Yaskawa INFORM job: R1_W03,5,7(0,0)OK-KM.JBI

/JOB
//NAME R1_W03,5,7(0,0)OK-KM
///FOLDERNAME SCIANA-NOWY-R2-KM
//POS
///NPOS 93,93,0,4,0,0
///TOOL 0
///POSTYPE PULSE
///PULSE
C00000=97801,-92951,-68020,42573,91743,-12282
C00001=188064,-59139,-49719,51220,48350,-5801
C00002=182482,-29523,-13831,58220,47542,-10694
C00003=186503,-14327,-833,57181,45005,-9773
C00004=186887,-13436,-157,57022,44797,-9650
C00005=187358,-18276,-5525,56185,44980,-9089
C00006=193250,-27913,-6363,58294,38967,-9969
C00007=199995,-16364,1412,54222,35645,-7165
C00008=199327,-15584,1994,54497,36056,-7364
C00009=199882,-17213,782,54333,35681,-7234
C00010=195511,-15034,9725,61255,35872,-11434
C00011=195511,-14418,11078,61887,35615,-11785
C00012=194782,-15937,9357,61766,36202,-11793
C00013=185148,-27392,-13403,56780,46393,-9588
C00014=194611,-49573,-33459,572,31924,-22077
C00015=195793,-42632,-27790,-753,32004,-21336
C00016=196651,-38308,-23003,-1749,31294,-20781
C00017=197052,-37261,-22343,-2197,31434,-20529
C00018=196235,-39864,-25459,-1248,31997,-21059
C00019=202582,-39238,-15691,-30047,22851,-6468
C00020=202582,-38747,-14553,-30589,22461,-6206
C00021=199520,-48265,-22642,-26019,21519,-8620
C00022=195597,-45769,-34616,8656,41829,-26358
C00023=205752,-37498,-18561,-12983,36783,-12907
C00024=204602,-36516,-17940,-11961,36728,-13544
C00025=195976,-39153,-18531,9623,35365,-26897
C00026=197793,-59286,-35313,7977,35152,-25873
C00027=213331,-48054,-41686,15165,61809,3623
C00028=205738,-19523,-29471,74829,71236,32232
C00029=212963,6142,-9202,90968,67126,41175
C00030=215317,9223,-6508,90706,65425,41155
C00031=216300,10496,-4975,90717,64708,41017
C00032=216595,12699,-3002,90716,64489,40979
C00033=216298,10454,-5417,90600,64716,41144
C00034=215808,9900,10687,95987,67227,42354
C00035=216745,9111,9989,96016,66542,42343
C00036=217921,4618,-10524,75178,67269,44249
C00037=217494,5264,-8626,75589,67333,43807
C00038=217735,7158,-6190,75755,67018,43579
C00039=220892,-10252,-22721,78838,53086,40871
C00040=217823,-16385,-27408,79730,55193,40452
C00041=213331,-48054,-41686,15165,61809,3623
C00042=211970,-37779,-14430,6801,34223,17849
C00043=210033,-36470,-13605,8545,34568,16753
C00044=209079,-35786,-13170,9389,34755,16221
C00045=208450,-36922,-14985,9824,35355,15936
C00046=209854,-36909,-13406,8784,34242,16610
C00047=205470,-32937,-11332,12488,35564,14251
C00048=204626,-32211,-10856,14325,36093,12193
C00049=199934,-27052,-7307,22881,40247,-2541
C00050=194869,-21825,-3734,26674,42807,-10107
C00051=213331,-48054,-41686,15165,61809,3623
C00052=227546,10998,5486,35197,58444,-54182
C00053=229778,13536,7768,34321,57451,-53482
C00054=230708,14716,8755,33927,57078,-53172
C00055=230020,15168,9251,34245,57291,-53423
C00056=230799,13170,6502,33684,57536,-52967
C00057=230268,3975,-668,31886,61076,-53028
C00058=230588,3390,-1036,31786,60892,-52943
C00059=229243,2878,-1594,32267,61468,-53362
C00060=231252,-39648,-4608,102791,21542,-67561
C00061=237258,-22465,5967,96694,21446,-64692
C00062=234738,-18513,13230,101595,23495,-67322
C00063=234315,-17869,14270,102096,23835,-67616
C00064=232289,-15111,19504,104909,25555,-69249
C00065=228307,-22326,11440,100405,28029,-67502
C00066=226911,810,-3337,33104,62378,-54110
C00067=213331,-48054,-41686,15165,61809,3623
C00068=211661,-57251,-25562,-55725,28615,-3338
C00069=209733,-56166,-24995,-54213,27635,-4283
C00070=209042,-55506,-24648,-53560,27321,-4674
C00071=207937,-56864,-25063,-53502,26430,-4804
C00072=210138,-56838,-26044,-54013,28046,-4347
C00073=213122,-57928,-25912,-64752,31046,-795
C00074=213758,-58111,-26008,-65027,31436,-589
C00075=219568,-60488,-27163,-67374,34939,1257
C00076=220810,-61245,-27594,-67808,35688,1626
C00077=221756,-61566,-27753,-68083,36274,1881
C00078=225369,-69260,-37480,-66382,39447,1288
C00079=205312,-39468,-16273,-14091,10779,-39550
C00080=202035,-29821,-9269,-1691,11105,-45367
C00081=201708,-29499,-9054,-507,11133,-45924
C00082=202005,-28855,-8724,-1550,11270,-45435
C00083=201579,-30109,-10785,-40,11885,-46143
C00084=201147,-30171,-8613,1607,10520,-46916
C00085=197038,-23502,-5168,15044,12246,-53254
C00086=191968,-16947,-326,28829,13963,-59823
C00087=192443,-23943,-5231,28759,13289,-59765
C00088=194260,-31922,-10655,25195,12023,-58034
C00089=194296,-50223,-21768,31420,9737,-60851
C00090=140544,-88669,-51716,31420,85002,-60851
C00091=29274,49299,-4686,19206,94492,-76966
C00092=-18103,108044,15339,14006,98532,-83827
BC00000=366006,1190719,810332
BC00001=395488,1192063,911452
BC00002=367626,1192063,911456
BC00003=367626,1192063,911456
BC00004=367626,1192063,911456
BC00005=367626,1192063,911456
BC00006=367626,1192063,911456
BC00007=367626,1192063,911456
BC00008=367626,1192063,911456
BC00009=367626,1192063,911456
BC00010=367626,1192063,911456
BC00011=367626,1192063,911456
BC00012=367626,1192063,911456
BC00013=367626,1192063,911456
BC00014=339752,1192063,946029
BC00015=339752,1192063,946029
BC00016=339752,1192063,946029
BC00017=339752,1192063,946029
BC00018=339752,1192063,946029
BC00019=339752,1192063,946029
BC00020=339752,1192063,946029
BC00021=339752,1192063,946029
BC00022=339752,1192063,946029
BC00023=339752,1192063,946029
BC00024=339752,1192063,946029
BC00025=339752,1192063,946029
BC00026=339752,1192063,946029
BC00027=343711,1192063,995389
BC00028=386489,1191732,674467
BC00029=396646,1191635,580346
BC00030=396646,1192063,571372
BC00031=396646,1192063,567782
BC00032=396646,1192063,567782
BC00033=396646,1192063,567782
BC00034=396646,1192063,632887
BC00035=396646,1192063,632887
BC00036=396646,1192063,632887
BC00037=396646,1192063,632887
BC00038=396646,1192063,632887
BC00039=396646,1192063,584688
BC00040=396646,1192063,601373
BC00041=343711,1192063,995389
BC00042=340575,1192063,995049
BC00043=334891,1192063,982003
BC00044=332050,1192063,975480
BC00045=332050,1192063,975480
BC00046=332050,1192063,975480
BC00047=341514,1192063,946969
BC00048=342419,1192063,946006
BC00049=345313,1192063,946292
BC00050=350589,1192063,932370
BC00051=343711,1192063,995389
BC00052=396646,1192063,884001
BC00053=396646,1192063,869517
BC00054=396646,1192063,862275
BC00055=396646,1192063,862275
BC00056=396646,1192063,862275
BC00057=396646,1192063,824652
BC00058=396646,1192062,824650
BC00059=396646,1192063,832496
BC00060=396646,1192063,832493
BC00061=396647,1192062,832490
BC00062=396647,1192062,832490
BC00063=396647,1192062,832490
BC00064=396647,1192062,832490
BC00065=396647,1192062,832490
BC00066=396646,1192063,848183
BC00067=343711,1192063,995389
BC00068=327217,1192063,959163
BC00069=320558,1192063,949782
BC00070=317895,1192063,946029
BC00071=317895,1192063,946029
BC00072=317895,1192063,946029
BC00073=315355,1192063,921524
BC00074=315345,1192063,914414
BC00075=315278,1192063,847952
BC00076=315266,1192063,833435
BC00077=317879,1192063,836911
BC00078=324411,1192063,845601
BC00079=373650,1192063,933673
BC00080=373828,1192063,927906
BC00081=366585,1192063,917035
BC00082=363688,1192063,912687
BC00083=363688,1192063,912687
BC00084=363688,1192063,912687
BC00085=363688,1192063,912687
BC00086=363688,1192063,912687
BC00087=366798,1192063,917263
BC00088=374041,1192063,928134
BC00089=374041,1192063,928134
BC00090=374041,1192063,928134
BC00091=213602,1191583,1029060
BC00092=114547,1272946,1072033
///POSTYPE BASE
///RECTAN
///RCONF 0,0,0,0,0,0,0,0,0,0,0,0,0,0,0,0,0,0,0,0,0,0,0,0
P00006=0.222,-3.123,-1.508,0.0000,0.0000,0.0000
P00021=-0.225,-6.128,-0.405,0.0000,0.0000,0.0000
P00024=0.145,-0.552,1.326,0.0000,0.0000,0.0000
P00027=-0.746,0.015,-9.096,0.0000,0.0000,0.0000
//INST
///DATE 2024/07/30 13:44
///ATTR SC,RW
///GROUP1 RB1,BS1
NOP
SFTOF
MOVJ C00000 BC00000 VJ=100.00
MOVJ C00001 BC00001 VJ=100.00
MOVJ C00002 BC00002 VJ=100.00
MOVL C00003 BC00003 V=60.0
REFP 3 C00004 BC00004
CALL JOB:SEARCH-R1
SET P021 P006
SFTON P021
MOVL C00005 BC00005 V=60.0
MOVL C00006 BC00006 V=100.0
MOVL C00007 BC00007 V=60.0
REFP 3 C00008 BC00008
CALL JOB:SEARCH-R1
SET P021 P006
SFTON P021
MOVL C00009 BC00009 V=60.0
MOVL C00010 BC00010 V=60.0
REFP 3 C00011 BC00011
CALL JOB:SEARCH-R1
SET P021 P006
SFTON P021
MOVL C00012 BC00012 V=60.0
MOVL C00013 BC00013 V=166.7
'Path S787 (for W405)
SFTOF
MOVL C00014 BC00014 V=100.0
MOVL C00015 BC00015 V=100.0
MOVL C00016 BC00016 V=60.0
REFP 3 C00017 BC00017
CALL JOB:SEARCH-R1
SET P027 P006
SFTON P027
MOVL C00018 BC00018 V=60.0
MOVL C00019 BC00019 V=60.0
REFP 3 C00020 BC00020
CALL JOB:SEARCH-R1
SET P027 P006
SFTON P027
MOVL C00021 BC00021 V=60.0
MOVL C00022 BC00022 V=100.0
MOVL C00023 BC00023 V=60.0
REFP 3 C00024 BC00024
CALL JOB:SEARCH-R1
SET P027 P006
SFTON P027
MOVL C00025 BC00025 V=60.0
MOVL C00026 BC00026 V=166.7
MOVJ C00027 BC00027 VJ=100.00
'Path S784 (for W404)
SFTOF
MOVJ C00028 BC00028 VJ=100.00
MOVJ C00029 BC00029 VJ=100.00
MOVJ C00030 BC00030 VJ=100.00
MOVL C00031 BC00031 V=100.0
REFP 3 C00032 BC00032
CALL JOB:SEARCH-R1
SET P024 P006
SFTON P024
MOVL C00033 BC00033 V=60.0
MOVL C00034 BC00034 V=60.0
REFP 3 C00035 BC00035
CALL JOB:SEARCH-R1
SET P024 P006
SFTON P024
MOVL C00036 BC00036 V=60.0
MOVL C00037 BC00037 V=60.0
REFP 3 C00038 BC00038
CALL JOB:SEARCH-R1
SET P024 P006
SFTON P024
MOVL C00039 BC00039 V=60.0
MOVL C00040 BC00040 V=166.7
MOVJ C00041 BC00041 VJ=100.00
'Path W402
SFTOF
SFTON P021
MOVJ C00042 BC00042 VJ=100.00
MOVJ C00043 BC00043 VJ=100.00
MOVL C00044 BC00044 V=100.0 PL=0
REFP 1 C00045 BC00045
REFP 2 C00046 BC00046
MACRO1 MJ#(0) ARGF10
ARCON
MOVL C00047 BC00047 V=13.3
MOVL C00048 BC00048 V=13.3
MOVL C00049 BC00049 V=13.3
MOVL C00050 BC00050 V=13.3
ARCOF
SFTOF
'
MOVJ C00051 BC00051 VJ=100.00
'
'Path W866
SFTOF
SFTON P024
MOVL C00052 BC00052 V=166.7
MOVL C00053 BC00053 V=166.7
MOVL C00054 BC00054 V=100.0 PL=0
REFP 1 C00055 BC00055
REFP 2 C00056 BC00056
MACRO1 MJ#(0) ARGF10
ARCON
MOVL C00057 BC00057 V=13.3
MOVL C00058 BC00058 V=11.7
ARCOF
MOVL C00059 BC00059 V=166.7
MOVL C00060 BC00060 V=166.7
MACRO1 MJ#(0) ARGF7
MOVL C00061 BC00061 V=166.7
ARCON
MOVL C00062 BC00062 V=11.7
MOVL C00063 BC00063 V=11.7
MOVL C00064 BC00064 V=11.7
ARCOF
MOVL C00065 BC00065 V=166.7
MOVL C00066 BC00066 V=166.7
SFTOF
'
MOVJ C00067 BC00067 VJ=100.00
'
'Path W405
SFTOF
SFTON P027
MOVL C00068 BC00068 V=166.7
MOVL C00069 BC00069 V=166.7
MOVL C00070 BC00070 V=100.0 PL=0
REFP 1 C00071 BC00071
REFP 2 C00072 BC00072
MACRO1 MJ#(0) ARGF10
ARCON
MOVL C00073 BC00073 V=13.3
MOVL C00074 BC00074 V=13.3
MOVL C00075 BC00075 V=13.3
MOVL C00076 BC00076 V=13.3
ARCOF
MOVL C00077 BC00077 V=166.7
MOVL C00078 BC00078 V=166.7
SFTOF
MOVJ C00079 BC00079 VJ=100.00
'Path W406
SFTOF
SFTON P027
MOVL C00080 BC00080 V=166.7
MOVL C00081 BC00081 V=166.7
MACRO1 MJ#(0) ARGF9
MOVL C00082 BC00082 V=100.0 PL=0
'WVON   ?????
ARCON
REFP 1 C00083 BC00083
REFP 2 C00084 BC00084
MACRO1 MJ#(0) ARGF7
MOVL C00085 BC00085 V=10.8
MOVL C00086 BC00086 V=10.8
ARCOF
WVOF
MOVL C00087 BC00087 V=166.7
MOVL C00088 BC00088 V=166.7
SFTOF
MOVJ C00089 BC00089 VJ=100.00
MOVJ C00090 BC00090 VJ=100.00
MOVJ C00091 BC00091 VJ=100.00
MOVJ C00092 BC00092 VJ=100.00
END
